// TIA Portal V17 export
// export: Created 2023-04-07T09:30:33.7447442Z, ExportSetting WithDefaults, DisplayName Totally Integrated Automation Portal, DisplayVersion V17 Update 4, DisplayName TIA Portal Openness, DisplayVersion V17 Update 4, DisplayName TIA Portal Version Control Interface, DisplayVersion V17, DisplayName STEP 7 Professional, DisplayVersion V17 Update 4, DisplayName STEP 7 Safety, DisplayVersion V17, DisplayName WinCC Professional, DisplayVersion V17 Update 4
FUNCTION "PCS W (S)_1" : Void   // FC44, LAD
TITLE = ModBus TCP for PCS Power Electronics
{ S7_Optimized_Access := 'TRUE' }
VERSION : 0.1
// stored: AutoNumber false, IsIECCheckEnabled false, SetENOAutomatically false, UDAEnableTagReadback false
   VAR_TEMP
      rSS1PacRef : Real;
      rSS2PacRef : Real;
      rSS1QacRef : Real;
      rSS2QacRef : Real;
      rSnHalfPE : Real;
      rQacRef : Real;
      uiQacRef : UInt;
   END_VAR
   VAR_TEMP   // added for the SCL form of the ladder/FBD networks
      _w1 : Bool;
   END_VAR
BEGIN

REGION Network 1: Function Modbus Client
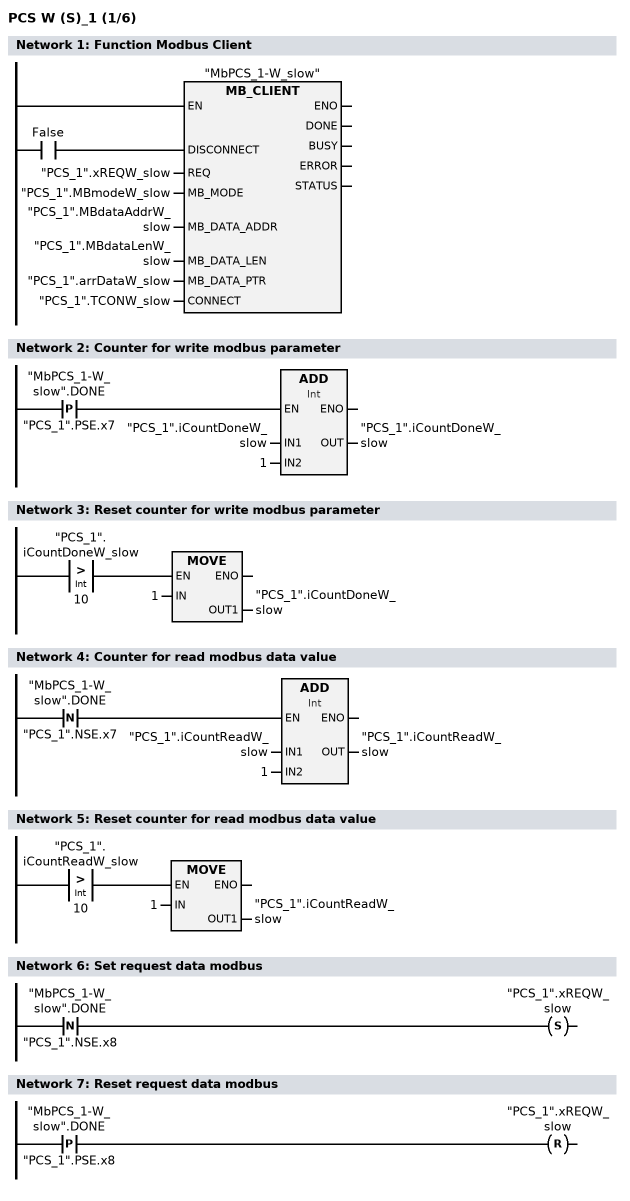
   RUNG wire#powerrail
      "MbPCS_1-W_slow".MB_CLIENT(DISCONNECT := wire#w1, REQ := "PCS_1".xREQW_slow, MB_MODE := "PCS_1".MBmodeW_slow, MB_DATA_ADDR := "PCS_1".MBdataAddrW_slow, MB_DATA_LEN := "PCS_1".MBdataLenW_slow, MB_DATA_PTR := "PCS_1".arrDataW_slow, CONNECT := "PCS_1".TCONW_slow, DONE =>, BUSY =>, ERROR =>, STATUS =>)
   END_RUNG
   RUNG wire#powerrail
      Contact( False )
   END_RUNG wire#w1
   // the same network as SCL:
   "MbPCS_1-W_slow"(DISCONNECT := False,   // MB_CLIENT
                    REQ := "PCS_1".xREQW_slow,
                    MB_MODE := "PCS_1".MBmodeW_slow,
                    MB_DATA_ADDR := "PCS_1".MBdataAddrW_slow,
                    MB_DATA_LEN := "PCS_1".MBdataLenW_slow,
                    MB_DATA_PTR := "PCS_1".arrDataW_slow,
                    CONNECT := "PCS_1".TCONW_slow);
END_REGION

REGION Network 2: Counter for write modbus parameter
   RUNG wire#powerrail
      P_Contact(operand := "MbPCS_1-W_slow".DONE, bit := "PCS_1".PSE.x7)
      { S7_Templates := "SrcType := Int" } Add(in1 := "PCS_1".iCountDoneW_slow, in2 := 1, out => "PCS_1".iCountDoneW_slow)
   END_RUNG
   // the same network as SCL:
   #_w1 := "MbPCS_1-W_slow".DONE AND NOT "PCS_1".PSE.x7;   // rising edge of "MbPCS_1-W_slow".DONE
   "PCS_1".PSE.x7 := "MbPCS_1-W_slow".DONE;
   IF #_w1 THEN "PCS_1".iCountDoneW_slow := "PCS_1".iCountDoneW_slow + 1; END_IF;
END_REGION

REGION Network 3: Reset counter for write modbus parameter
   RUNG wire#powerrail
      { S7_Templates := "SrcType := Int" } GT_Contact(in1 := "PCS_1".iCountDoneW_slow, in2 := 10)
      Move(in := 1, out1 => "PCS_1".iCountDoneW_slow)
   END_RUNG
   // the same network as SCL:
   IF "PCS_1".iCountDoneW_slow > 10 THEN "PCS_1".iCountDoneW_slow := 1; END_IF;
END_REGION

REGION Network 4: Counter for read modbus data value
   RUNG wire#powerrail
      N_Contact(operand := "MbPCS_1-W_slow".DONE, bit := "PCS_1".NSE.x7)
      { S7_Templates := "SrcType := Int" } Add(in1 := "PCS_1".iCountReadW_slow, in2 := 1, out => "PCS_1".iCountReadW_slow)
   END_RUNG
   // the same network as SCL:
   #_w1 := NOT "MbPCS_1-W_slow".DONE AND "PCS_1".NSE.x7;   // falling edge of "MbPCS_1-W_slow".DONE
   "PCS_1".NSE.x7 := "MbPCS_1-W_slow".DONE;
   IF #_w1 THEN "PCS_1".iCountReadW_slow := "PCS_1".iCountReadW_slow + 1; END_IF;
END_REGION

REGION Network 5: Reset counter for read modbus data value
   RUNG wire#powerrail
      { S7_Templates := "SrcType := Int" } GT_Contact(in1 := "PCS_1".iCountReadW_slow, in2 := 10)
      Move(in := 1, out1 => "PCS_1".iCountReadW_slow)
   END_RUNG
   // the same network as SCL:
   IF "PCS_1".iCountReadW_slow > 10 THEN "PCS_1".iCountReadW_slow := 1; END_IF;
END_REGION

REGION Network 6: Set request data modbus
   RUNG wire#powerrail
      N_Contact(operand := "MbPCS_1-W_slow".DONE, bit := "PCS_1".NSE.x8)
      S_Coil( "PCS_1".xREQW_slow )
   END_RUNG
   // the same network as SCL:
   #_w1 := NOT "MbPCS_1-W_slow".DONE AND "PCS_1".NSE.x8;   // falling edge of "MbPCS_1-W_slow".DONE
   "PCS_1".NSE.x8 := "MbPCS_1-W_slow".DONE;
   IF #_w1 THEN "PCS_1".xREQW_slow := TRUE; END_IF;
END_REGION

REGION Network 7: Reset request data modbus
   RUNG wire#powerrail
      P_Contact(operand := "MbPCS_1-W_slow".DONE, bit := "PCS_1".PSE.x8)
      R_Coil( "PCS_1".xREQW_slow )
   END_RUNG
   // the same network as SCL:
   #_w1 := "MbPCS_1-W_slow".DONE AND NOT "PCS_1".PSE.x8;   // rising edge of "MbPCS_1-W_slow".DONE
   "PCS_1".PSE.x8 := "MbPCS_1-W_slow".DONE;
   IF #_w1 THEN "PCS_1".xREQW_slow := FALSE; END_IF;
END_REGION

REGION Network 9: Write W_Block1 parameter - pwd to check
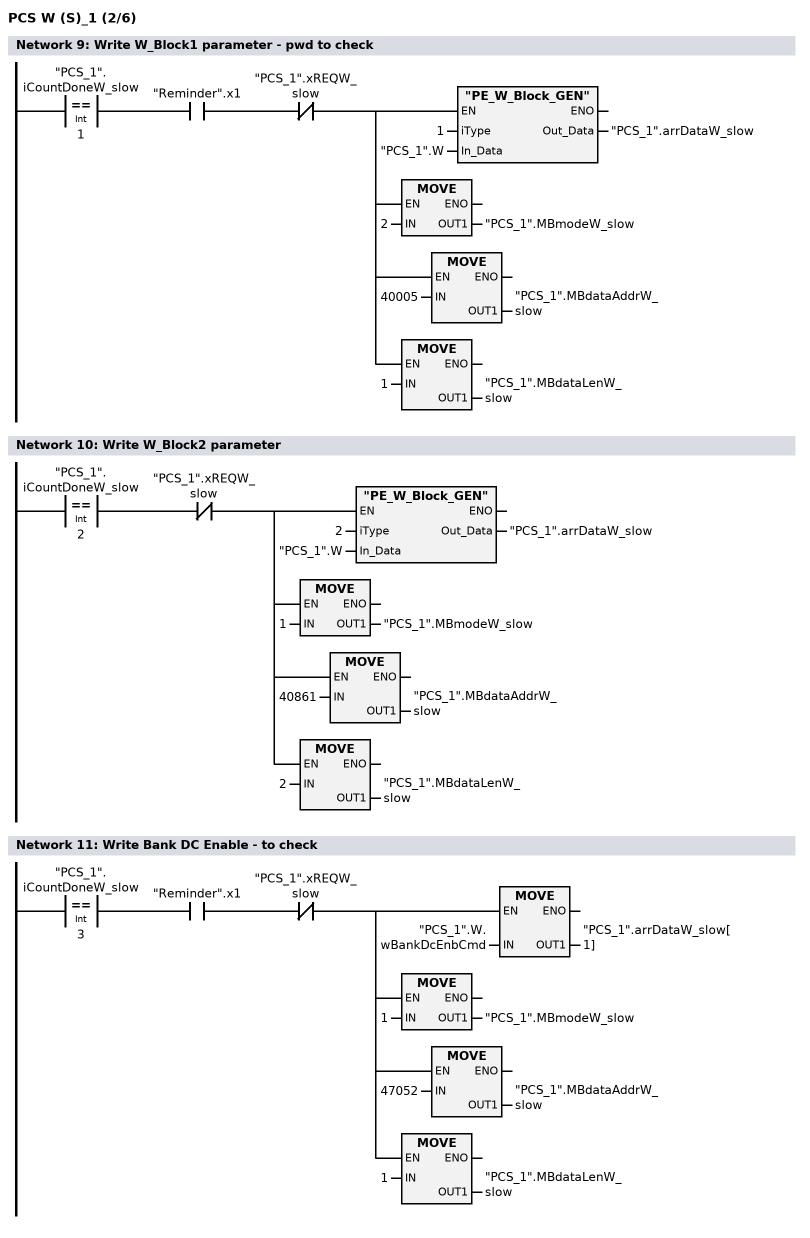
   RUNG wire#powerrail
      { S7_Templates := "SrcType := Int" } EQ_Contact(in1 := "PCS_1".iCountDoneW_slow, in2 := 1)
      Contact( "Reminder".x1 )
      I_Contact( "PCS_1".xREQW_slow )
      wire#w1
      "PE_W_Block_GEN"(iType := 1, In_Data := "PCS_1".W, Out_Data => "PCS_1".arrDataW_slow)
   END_RUNG
   RUNG wire#w1
      Move(in := 2, out1 => "PCS_1".MBmodeW_slow)
   END_RUNG
   RUNG wire#w1
      Move(in := 40005, out1 => "PCS_1".MBdataAddrW_slow)
   END_RUNG
   RUNG wire#w1
      Move(in := 1, out1 => "PCS_1".MBdataLenW_slow)
   END_RUNG
   // the same network as SCL:
   #_w1 := ("PCS_1".iCountDoneW_slow = 1) AND "Reminder".x1 AND NOT "PCS_1".xREQW_slow;
   IF #_w1 THEN
       "PE_W_Block_GEN"(iType := 1, In_Data := "PCS_1".W, Out_Data => "PCS_1".arrDataW_slow);
       "PCS_1".MBmodeW_slow := 2;
       "PCS_1".MBdataAddrW_slow := 40005;
       "PCS_1".MBdataLenW_slow := 1;
   END_IF;
END_REGION

REGION Network 10: Write W_Block2 parameter
   RUNG wire#powerrail
      { S7_Templates := "SrcType := Int" } EQ_Contact(in1 := "PCS_1".iCountDoneW_slow, in2 := 2)
      I_Contact( "PCS_1".xREQW_slow )
      wire#w1
      "PE_W_Block_GEN"(iType := 2, In_Data := "PCS_1".W, Out_Data => "PCS_1".arrDataW_slow)
   END_RUNG
   RUNG wire#w1
      Move(in := 1, out1 => "PCS_1".MBmodeW_slow)
   END_RUNG
   RUNG wire#w1
      Move(in := 40861, out1 => "PCS_1".MBdataAddrW_slow)
   END_RUNG
   RUNG wire#w1
      Move(in := 2, out1 => "PCS_1".MBdataLenW_slow)
   END_RUNG
   // the same network as SCL:
   #_w1 := ("PCS_1".iCountDoneW_slow = 2) AND NOT "PCS_1".xREQW_slow;
   IF #_w1 THEN
       "PE_W_Block_GEN"(iType := 2, In_Data := "PCS_1".W, Out_Data => "PCS_1".arrDataW_slow);
       "PCS_1".MBmodeW_slow := 1;
       "PCS_1".MBdataAddrW_slow := 40861;
       "PCS_1".MBdataLenW_slow := 2;
   END_IF;
END_REGION

REGION Network 11: Write Bank DC Enable - to check
   RUNG wire#powerrail
      { S7_Templates := "SrcType := Int" } EQ_Contact(in1 := "PCS_1".iCountDoneW_slow, in2 := 3)
      Contact( "Reminder".x1 )
      I_Contact( "PCS_1".xREQW_slow )
      wire#w1
      Move(in := "PCS_1".W.wBankDcEnbCmd, out1 => "PCS_1".arrDataW_slow[1])
   END_RUNG
   RUNG wire#w1
      Move(in := 1, out1 => "PCS_1".MBmodeW_slow)
   END_RUNG
   RUNG wire#w1
      Move(in := 47052, out1 => "PCS_1".MBdataAddrW_slow)
   END_RUNG
   RUNG wire#w1
      Move(in := 1, out1 => "PCS_1".MBdataLenW_slow)
   END_RUNG
   // the same network as SCL:
   IF ("PCS_1".iCountDoneW_slow = 3) AND "Reminder".x1 AND NOT "PCS_1".xREQW_slow THEN
       "PCS_1".arrDataW_slow[1] := "PCS_1".W.wBankDcEnbCmd;
       "PCS_1".MBmodeW_slow := 1;
       "PCS_1".MBdataAddrW_slow := 47052;
       "PCS_1".MBdataLenW_slow := 1;
   END_IF;
END_REGION

REGION Network 12: Write Qac Reference
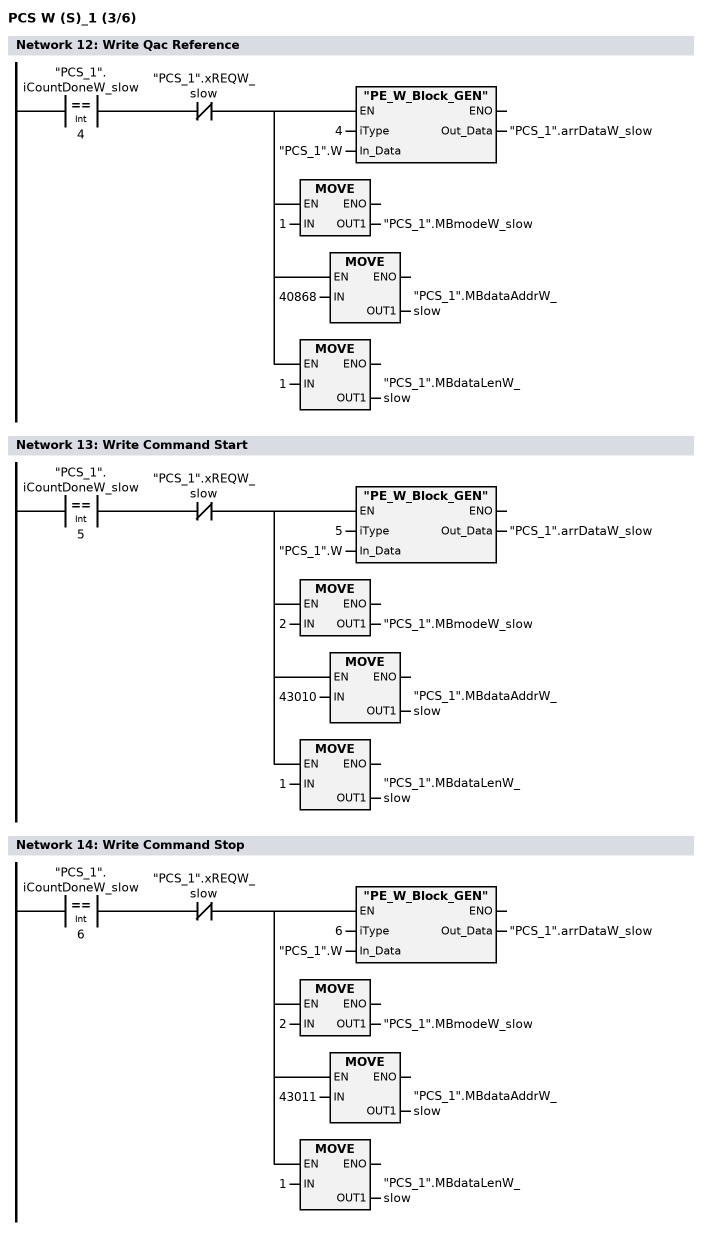
   RUNG wire#powerrail
      { S7_Templates := "SrcType := Int" } EQ_Contact(in1 := "PCS_1".iCountDoneW_slow, in2 := 4)
      I_Contact( "PCS_1".xREQW_slow )
      wire#w1
      "PE_W_Block_GEN"(iType := 4, In_Data := "PCS_1".W, Out_Data => "PCS_1".arrDataW_slow)
   END_RUNG
   RUNG wire#w1
      Move(in := 1, out1 => "PCS_1".MBmodeW_slow)
   END_RUNG
   RUNG wire#w1
      Move(in := 40868, out1 => "PCS_1".MBdataAddrW_slow)
   END_RUNG
   RUNG wire#w1
      Move(in := 1, out1 => "PCS_1".MBdataLenW_slow)
   END_RUNG
   // the same network as SCL:
   #_w1 := ("PCS_1".iCountDoneW_slow = 4) AND NOT "PCS_1".xREQW_slow;
   IF #_w1 THEN
       "PE_W_Block_GEN"(iType := 4, In_Data := "PCS_1".W, Out_Data => "PCS_1".arrDataW_slow);
       "PCS_1".MBmodeW_slow := 1;
       "PCS_1".MBdataAddrW_slow := 40868;
       "PCS_1".MBdataLenW_slow := 1;
   END_IF;
END_REGION

REGION Network 13: Write Command Start
   RUNG wire#powerrail
      { S7_Templates := "SrcType := Int" } EQ_Contact(in1 := "PCS_1".iCountDoneW_slow, in2 := 5)
      I_Contact( "PCS_1".xREQW_slow )
      wire#w1
      "PE_W_Block_GEN"(iType := 5, In_Data := "PCS_1".W, Out_Data => "PCS_1".arrDataW_slow)
   END_RUNG
   RUNG wire#w1
      Move(in := 2, out1 => "PCS_1".MBmodeW_slow)
   END_RUNG
   RUNG wire#w1
      Move(in := 43010, out1 => "PCS_1".MBdataAddrW_slow)
   END_RUNG
   RUNG wire#w1
      Move(in := 1, out1 => "PCS_1".MBdataLenW_slow)
   END_RUNG
   // the same network as SCL:
   #_w1 := ("PCS_1".iCountDoneW_slow = 5) AND NOT "PCS_1".xREQW_slow;
   IF #_w1 THEN
       "PE_W_Block_GEN"(iType := 5, In_Data := "PCS_1".W, Out_Data => "PCS_1".arrDataW_slow);
       "PCS_1".MBmodeW_slow := 2;
       "PCS_1".MBdataAddrW_slow := 43010;
       "PCS_1".MBdataLenW_slow := 1;
   END_IF;
END_REGION

REGION Network 14: Write Command Stop
   RUNG wire#powerrail
      { S7_Templates := "SrcType := Int" } EQ_Contact(in1 := "PCS_1".iCountDoneW_slow, in2 := 6)
      I_Contact( "PCS_1".xREQW_slow )
      wire#w1
      "PE_W_Block_GEN"(iType := 6, In_Data := "PCS_1".W, Out_Data => "PCS_1".arrDataW_slow)
   END_RUNG
   RUNG wire#w1
      Move(in := 2, out1 => "PCS_1".MBmodeW_slow)
   END_RUNG
   RUNG wire#w1
      Move(in := 43011, out1 => "PCS_1".MBdataAddrW_slow)
   END_RUNG
   RUNG wire#w1
      Move(in := 1, out1 => "PCS_1".MBdataLenW_slow)
   END_RUNG
   // the same network as SCL:
   #_w1 := ("PCS_1".iCountDoneW_slow = 6) AND NOT "PCS_1".xREQW_slow;
   IF #_w1 THEN
       "PE_W_Block_GEN"(iType := 6, In_Data := "PCS_1".W, Out_Data => "PCS_1".arrDataW_slow);
       "PCS_1".MBmodeW_slow := 2;
       "PCS_1".MBdataAddrW_slow := 43011;
       "PCS_1".MBdataLenW_slow := 1;
   END_IF;
END_REGION

REGION Network 15: Write Command Reset Fault
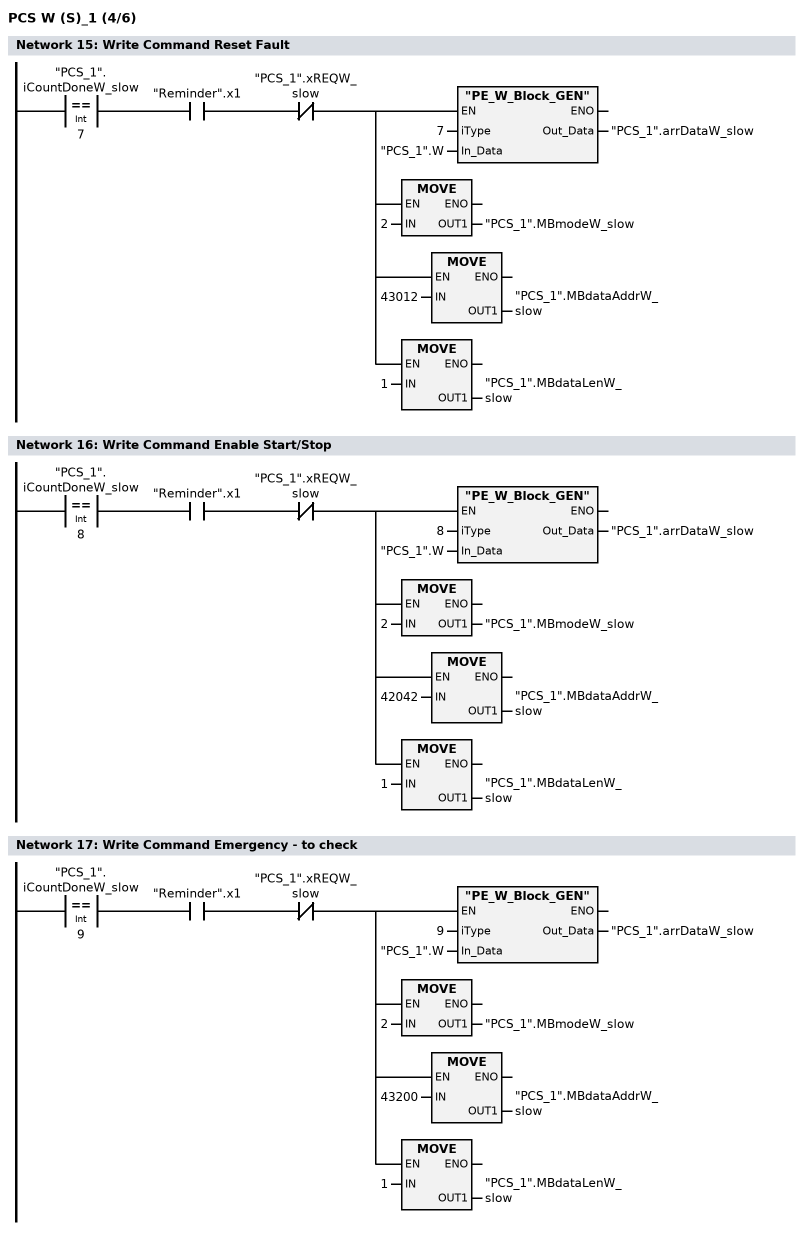
   RUNG wire#powerrail
      { S7_Templates := "SrcType := Int" } EQ_Contact(in1 := "PCS_1".iCountDoneW_slow, in2 := 7)
      Contact( "Reminder".x1 )
      I_Contact( "PCS_1".xREQW_slow )
      wire#w1
      "PE_W_Block_GEN"(iType := 7, In_Data := "PCS_1".W, Out_Data => "PCS_1".arrDataW_slow)
   END_RUNG
   RUNG wire#w1
      Move(in := 2, out1 => "PCS_1".MBmodeW_slow)
   END_RUNG
   RUNG wire#w1
      Move(in := 43012, out1 => "PCS_1".MBdataAddrW_slow)
   END_RUNG
   RUNG wire#w1
      Move(in := 1, out1 => "PCS_1".MBdataLenW_slow)
   END_RUNG
   // the same network as SCL:
   #_w1 := ("PCS_1".iCountDoneW_slow = 7) AND "Reminder".x1 AND NOT "PCS_1".xREQW_slow;
   IF #_w1 THEN
       "PE_W_Block_GEN"(iType := 7, In_Data := "PCS_1".W, Out_Data => "PCS_1".arrDataW_slow);
       "PCS_1".MBmodeW_slow := 2;
       "PCS_1".MBdataAddrW_slow := 43012;
       "PCS_1".MBdataLenW_slow := 1;
   END_IF;
END_REGION

REGION Network 16: Write Command Enable Start/Stop
   RUNG wire#powerrail
      { S7_Templates := "SrcType := Int" } EQ_Contact(in1 := "PCS_1".iCountDoneW_slow, in2 := 8)
      Contact( "Reminder".x1 )
      I_Contact( "PCS_1".xREQW_slow )
      wire#w1
      "PE_W_Block_GEN"(iType := 8, In_Data := "PCS_1".W, Out_Data => "PCS_1".arrDataW_slow)
   END_RUNG
   RUNG wire#w1
      Move(in := 2, out1 => "PCS_1".MBmodeW_slow)
   END_RUNG
   RUNG wire#w1
      Move(in := 42042, out1 => "PCS_1".MBdataAddrW_slow)
   END_RUNG
   RUNG wire#w1
      Move(in := 1, out1 => "PCS_1".MBdataLenW_slow)
   END_RUNG
   // the same network as SCL:
   #_w1 := ("PCS_1".iCountDoneW_slow = 8) AND "Reminder".x1 AND NOT "PCS_1".xREQW_slow;
   IF #_w1 THEN
       "PE_W_Block_GEN"(iType := 8, In_Data := "PCS_1".W, Out_Data => "PCS_1".arrDataW_slow);
       "PCS_1".MBmodeW_slow := 2;
       "PCS_1".MBdataAddrW_slow := 42042;
       "PCS_1".MBdataLenW_slow := 1;
   END_IF;
END_REGION

REGION Network 17: Write Command Emergency - to check
   RUNG wire#powerrail
      { S7_Templates := "SrcType := Int" } EQ_Contact(in1 := "PCS_1".iCountDoneW_slow, in2 := 9)
      Contact( "Reminder".x1 )
      I_Contact( "PCS_1".xREQW_slow )
      wire#w1
      "PE_W_Block_GEN"(iType := 9, In_Data := "PCS_1".W, Out_Data => "PCS_1".arrDataW_slow)
   END_RUNG
   RUNG wire#w1
      Move(in := 2, out1 => "PCS_1".MBmodeW_slow)
   END_RUNG
   RUNG wire#w1
      Move(in := 43200, out1 => "PCS_1".MBdataAddrW_slow)
   END_RUNG
   RUNG wire#w1
      Move(in := 1, out1 => "PCS_1".MBdataLenW_slow)
   END_RUNG
   // the same network as SCL:
   #_w1 := ("PCS_1".iCountDoneW_slow = 9) AND "Reminder".x1 AND NOT "PCS_1".xREQW_slow;
   IF #_w1 THEN
       "PE_W_Block_GEN"(iType := 9, In_Data := "PCS_1".W, Out_Data => "PCS_1".arrDataW_slow);
       "PCS_1".MBmodeW_slow := 2;
       "PCS_1".MBdataAddrW_slow := 43200;
       "PCS_1".MBdataLenW_slow := 1;
   END_IF;
END_REGION

REGION Network 18: Write WatchDog - to check
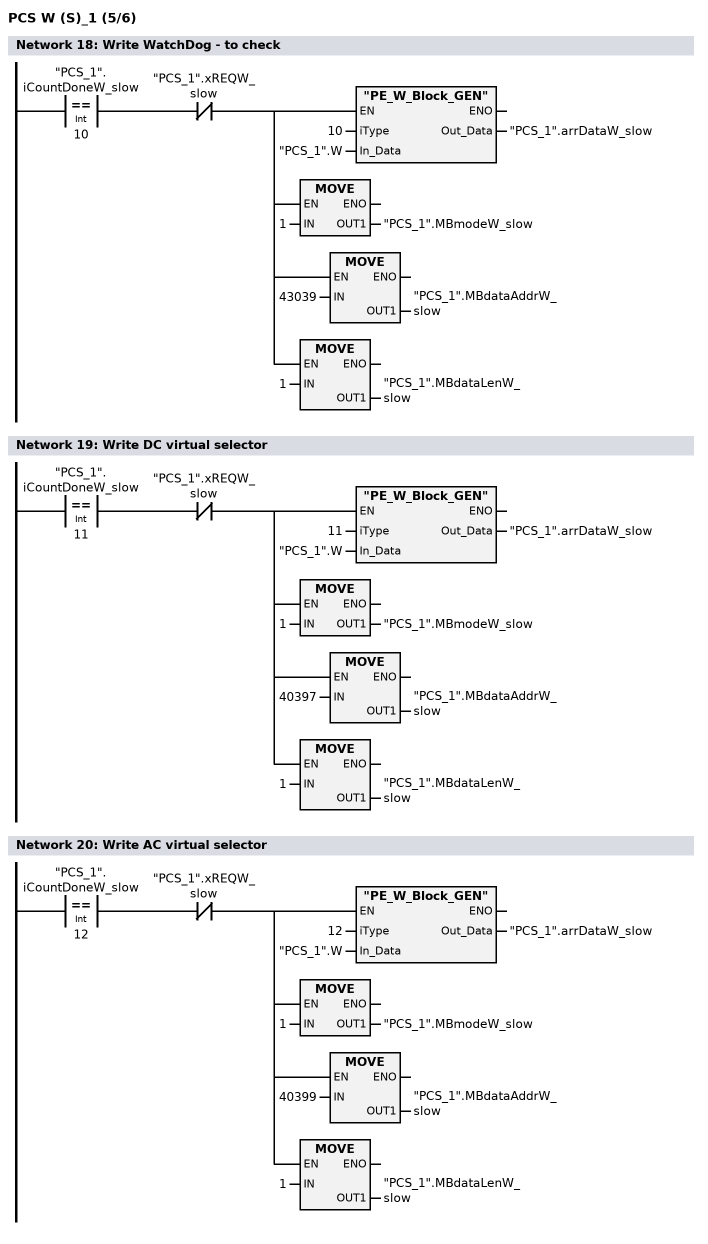
   RUNG wire#powerrail
      { S7_Templates := "SrcType := Int" } EQ_Contact(in1 := "PCS_1".iCountDoneW_slow, in2 := 10)
      I_Contact( "PCS_1".xREQW_slow )
      wire#w1
      "PE_W_Block_GEN"(iType := 10, In_Data := "PCS_1".W, Out_Data => "PCS_1".arrDataW_slow)
   END_RUNG
   RUNG wire#w1
      Move(in := 1, out1 => "PCS_1".MBmodeW_slow)
   END_RUNG
   RUNG wire#w1
      Move(in := 43039, out1 => "PCS_1".MBdataAddrW_slow)
   END_RUNG
   RUNG wire#w1
      Move(in := 1, out1 => "PCS_1".MBdataLenW_slow)
   END_RUNG
   // the same network as SCL:
   #_w1 := ("PCS_1".iCountDoneW_slow = 10) AND NOT "PCS_1".xREQW_slow;
   IF #_w1 THEN
       "PE_W_Block_GEN"(iType := 10, In_Data := "PCS_1".W, Out_Data => "PCS_1".arrDataW_slow);
       "PCS_1".MBmodeW_slow := 1;
       "PCS_1".MBdataAddrW_slow := 43039;
       "PCS_1".MBdataLenW_slow := 1;
   END_IF;
END_REGION

REGION Network 19: Write DC virtual selector
   RUNG wire#powerrail
      { S7_Templates := "SrcType := Int" } EQ_Contact(in1 := "PCS_1".iCountDoneW_slow, in2 := 11)
      I_Contact( "PCS_1".xREQW_slow )
      wire#w1
      "PE_W_Block_GEN"(iType := 11, In_Data := "PCS_1".W, Out_Data => "PCS_1".arrDataW_slow)
   END_RUNG
   RUNG wire#w1
      Move(in := 1, out1 => "PCS_1".MBmodeW_slow)
   END_RUNG
   RUNG wire#w1
      Move(in := 40397, out1 => "PCS_1".MBdataAddrW_slow)
   END_RUNG
   RUNG wire#w1
      Move(in := 1, out1 => "PCS_1".MBdataLenW_slow)
   END_RUNG
   // the same network as SCL:
   #_w1 := ("PCS_1".iCountDoneW_slow = 11) AND NOT "PCS_1".xREQW_slow;
   IF #_w1 THEN
       "PE_W_Block_GEN"(iType := 11, In_Data := "PCS_1".W, Out_Data => "PCS_1".arrDataW_slow);
       "PCS_1".MBmodeW_slow := 1;
       "PCS_1".MBdataAddrW_slow := 40397;
       "PCS_1".MBdataLenW_slow := 1;
   END_IF;
END_REGION

REGION Network 20: Write AC virtual selector
   RUNG wire#powerrail
      { S7_Templates := "SrcType := Int" } EQ_Contact(in1 := "PCS_1".iCountDoneW_slow, in2 := 12)
      I_Contact( "PCS_1".xREQW_slow )
      wire#w1
      "PE_W_Block_GEN"(iType := 12, In_Data := "PCS_1".W, Out_Data => "PCS_1".arrDataW_slow)
   END_RUNG
   RUNG wire#w1
      Move(in := 1, out1 => "PCS_1".MBmodeW_slow)
   END_RUNG
   RUNG wire#w1
      Move(in := 40399, out1 => "PCS_1".MBdataAddrW_slow)
   END_RUNG
   RUNG wire#w1
      Move(in := 1, out1 => "PCS_1".MBdataLenW_slow)
   END_RUNG
   // the same network as SCL:
   #_w1 := ("PCS_1".iCountDoneW_slow = 12) AND NOT "PCS_1".xREQW_slow;
   IF #_w1 THEN
       "PE_W_Block_GEN"(iType := 12, In_Data := "PCS_1".W, Out_Data => "PCS_1".arrDataW_slow);
       "PCS_1".MBmodeW_slow := 1;
       "PCS_1".MBdataAddrW_slow := 40399;
       "PCS_1".MBdataLenW_slow := 1;
   END_IF;
END_REGION

REGION Network 21: Write General selector
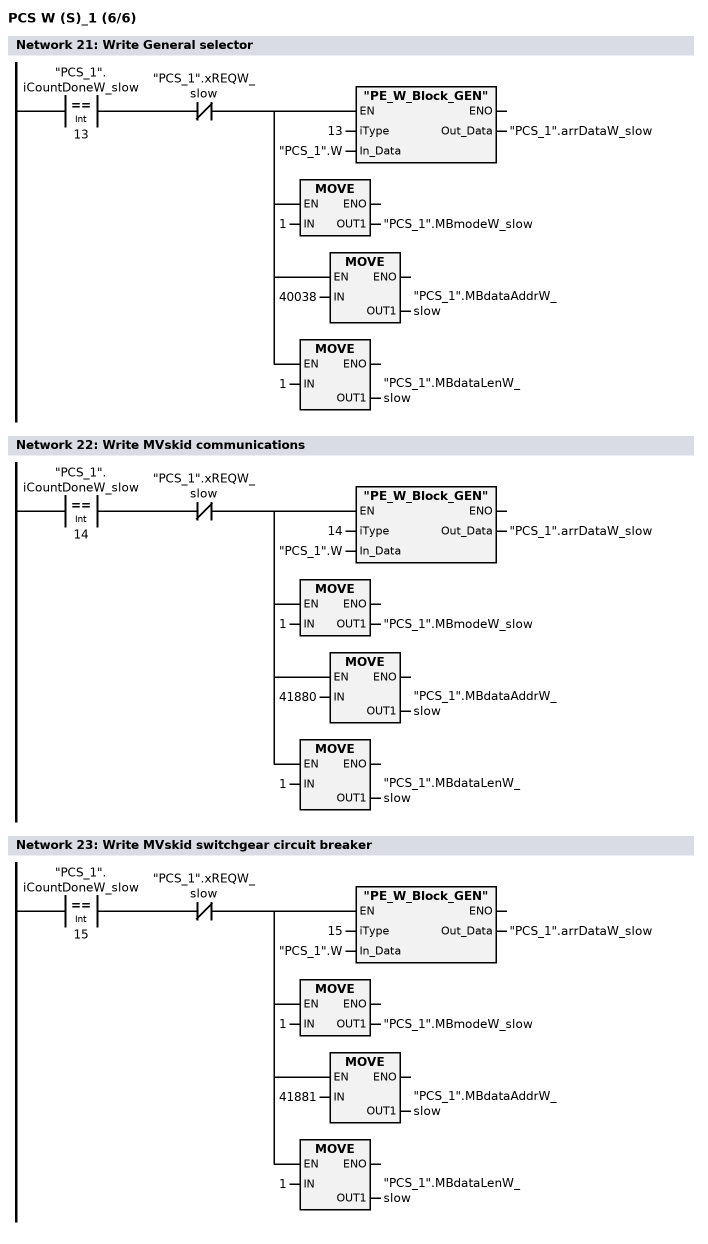
   RUNG wire#powerrail
      { S7_Templates := "SrcType := Int" } EQ_Contact(in1 := "PCS_1".iCountDoneW_slow, in2 := 13)
      I_Contact( "PCS_1".xREQW_slow )
      wire#w1
      "PE_W_Block_GEN"(iType := 13, In_Data := "PCS_1".W, Out_Data => "PCS_1".arrDataW_slow)
   END_RUNG
   RUNG wire#w1
      Move(in := 1, out1 => "PCS_1".MBmodeW_slow)
   END_RUNG
   RUNG wire#w1
      Move(in := 40038, out1 => "PCS_1".MBdataAddrW_slow)
   END_RUNG
   RUNG wire#w1
      Move(in := 1, out1 => "PCS_1".MBdataLenW_slow)
   END_RUNG
   // the same network as SCL:
   #_w1 := ("PCS_1".iCountDoneW_slow = 13) AND NOT "PCS_1".xREQW_slow;
   IF #_w1 THEN
       "PE_W_Block_GEN"(iType := 13, In_Data := "PCS_1".W, Out_Data => "PCS_1".arrDataW_slow);
       "PCS_1".MBmodeW_slow := 1;
       "PCS_1".MBdataAddrW_slow := 40038;
       "PCS_1".MBdataLenW_slow := 1;
   END_IF;
END_REGION

REGION Network 22: Write MVskid communications
   RUNG wire#powerrail
      { S7_Templates := "SrcType := Int" } EQ_Contact(in1 := "PCS_1".iCountDoneW_slow, in2 := 14)
      I_Contact( "PCS_1".xREQW_slow )
      wire#w1
      "PE_W_Block_GEN"(iType := 14, In_Data := "PCS_1".W, Out_Data => "PCS_1".arrDataW_slow)
   END_RUNG
   RUNG wire#w1
      Move(in := 1, out1 => "PCS_1".MBmodeW_slow)
   END_RUNG
   RUNG wire#w1
      Move(in := 41880, out1 => "PCS_1".MBdataAddrW_slow)
   END_RUNG
   RUNG wire#w1
      Move(in := 1, out1 => "PCS_1".MBdataLenW_slow)
   END_RUNG
   // the same network as SCL:
   #_w1 := ("PCS_1".iCountDoneW_slow = 14) AND NOT "PCS_1".xREQW_slow;
   IF #_w1 THEN
       "PE_W_Block_GEN"(iType := 14, In_Data := "PCS_1".W, Out_Data => "PCS_1".arrDataW_slow);
       "PCS_1".MBmodeW_slow := 1;
       "PCS_1".MBdataAddrW_slow := 41880;
       "PCS_1".MBdataLenW_slow := 1;
   END_IF;
END_REGION

REGION Network 23: Write MVskid switchgear circuit breaker
   RUNG wire#powerrail
      { S7_Templates := "SrcType := Int" } EQ_Contact(in1 := "PCS_1".iCountDoneW_slow, in2 := 15)
      I_Contact( "PCS_1".xREQW_slow )
      wire#w1
      "PE_W_Block_GEN"(iType := 15, In_Data := "PCS_1".W, Out_Data => "PCS_1".arrDataW_slow)
   END_RUNG
   RUNG wire#w1
      Move(in := 1, out1 => "PCS_1".MBmodeW_slow)
   END_RUNG
   RUNG wire#w1
      Move(in := 41881, out1 => "PCS_1".MBdataAddrW_slow)
   END_RUNG
   RUNG wire#w1
      Move(in := 1, out1 => "PCS_1".MBdataLenW_slow)
   END_RUNG
   // the same network as SCL:
   #_w1 := ("PCS_1".iCountDoneW_slow = 15) AND NOT "PCS_1".xREQW_slow;
   IF #_w1 THEN
       "PE_W_Block_GEN"(iType := 15, In_Data := "PCS_1".W, Out_Data => "PCS_1".arrDataW_slow);
       "PCS_1".MBmodeW_slow := 1;
       "PCS_1".MBdataAddrW_slow := 41881;
       "PCS_1".MBdataLenW_slow := 1;
   END_IF;
END_REGION
END_FUNCTION
